// TIA Portal V20 export
VAR_GLOBAL   // PLC tag table "CABIN"
   cabinDoorControlCh1 AT %I400.0 : Bool;   // Cabin door control switch Channel 1
   cabinDoorControlCh2 AT %I400.4 : Bool;   // Cabin door control switch Channel 2
   cabinDoorControlCh1VS AT %I401.0 : Bool;   // Cabin door control switch Channel 1 supply
   cabinDoorControlCh2VS AT %I401.4 : Bool;   // Cabin door control switch Channel 2 supply
   cabinDoorControlFb AT %I450.0 : Bool;   // Cabin door control switch Feedback
   cbHMIPcSupply AT %I450.1 : Bool;   // HMI, PC supply CB Feedback
   cbOperatorChair24VdcSupply AT %I450.2 : Bool;   // Operator chair 24VDC supply CB Feedback
   "cbCabin400VLoads(1)" AT %I450.3 : Bool;   // Cabin 400V loads CB Feedback
   cbCabin230VCircuits AT %I450.4 : Bool;   // Cabin 230V circuits CB Feedback
   cbCabinSignalLights AT %I450.5 : Bool;   // Cabin signal lights CB
   cbWindshieldWiper AT %I452.1 : Bool;   // Windshield wiper CB Feedback
   cbWindshieldWaterPump AT %I452.2 : Bool;   // Windshield water pump CB Feedback
   cbRoofWindshieldWiper AT %I452.3 : Bool;   // Roof windshield wiper CB Feedback
   cbRoofWindshieldWaterPump AT %I452.4 : Bool;   // Roof windshield water pump CB Feedback
   cbCabinAC AT %I452.6 : Bool;   // Cabin AC CB Feedback
   cbCabinSockets AT %I452.7 : Bool;   // Cabin sockets CBs Feedback
   cbCabinHeating400Vrcb AT %I453.0 : Bool;   // Cabin heating 400V RCB Feedback
   cbCabinHeaters AT %I453.1 : Bool;   // Cabin heaters CBs Feedback
   cb24CabinFanPs AT %I453.2 : Bool;   // 24VDC cabin fan PS CB Feedback
   cabinFanPs24Ok AT %I453.3 : Bool;   // 24VDC cabin fan PS OK
   cbCabinIllumination AT %I453.4 : Bool;   // Cabin illumination CBs Feedback
   footSwitch AT %I453.5 : Bool;   // Footswitch Feedback
   indSpreaderLanded AT %Q450.0 : Bool;   // Spreader status indication Landed
   indSpreaderLocked AT %Q450.1 : Bool;   // Spreader status indication Locked
   indSpreaderUnlocked AT %Q450.2 : Bool;   // Spreader status indication Unlocked
   indSpreaderOverload AT %Q450.3 : Bool;   // Spreader status indication Overload
   indSpreaderTwinDown AT %Q450.4 : Bool;   // Spreader status indication Twin down
   indSpreaderSnagLoad AT %Q450.5 : Bool;   // Spreader status indication Snag load
   windshieldWiperStart AT %Q450.6 : Bool;   // Windshield wiper control relay
   windshieldPumpStart AT %Q450.7 : Bool;   // Windshield water pump control relay
   roofWindshieldWiperStart AT %Q451.0 : Bool;   // Roof windshield wiper control relay
   roofWindshieldPumpStart AT %Q451.1 : Bool;   // Roof windshield water pump control relay
   indCabinRedC1 AT %Q451.2 : Bool;   // Cabin signal light Red C1 mode relay
   indCabinRedC2 AT %Q451.3 : Bool;   // Cabin signal light Red C2 mode relay
   indCabinGreenC1 AT %Q451.4 : Bool;   // Cabin signal light Green C1 mode relay
   indCabinGreenC2 AT %Q451.5 : Bool;   // Cabin signal light Green C2 mode relay
   indCabinBlueC1 AT %Q451.6 : Bool;   // Cabin signal light Blue C1 mode relay
   indCabinBlueC2 AT %Q451.7 : Bool;   // Cabin signal light Blue C2 mode relay
   mTEMP_LOGIC1 AT %M1.1 : Bool;
   mTEMP_LOGIC0 AT %M1.0 : Bool;
   btnEmStopCabinCh2 AT %I400.5 : Bool;   // Emergency Stop pushbutton Channel 2
   btnEmStopCabinCh2VS AT %I401.5 : Bool;   // Emergency Stop pushbutton Channel 2 Supply
   btnEmStopCabinCh1 AT %I400.1 : Bool;   // Emergency Stop pushbutton Channel 1
   btnEmStopCabinCh1VS AT %I401.1 : Bool;   // Emergency Stop pushbutton Channel 1 Supply
   "washingPS24Ok(1)" AT %I452.5 : Bool;   // 24VDC washing PS OK
   "cb24WashingPS(1)" AT %I452.0 : Bool;   // 24VDC washing PS CB Feedback
END_VAR
